(* IEC 61131-3 sources: volt/packages/volt-lsp-iec/test-corpus/bakon-nano/Device/Plc Logic/Application/Library Manager/(unresolved)/visu interfaces, 19 files *)

(* ---- RECIPE_FILEPARAMETERS.dut ---- *)
TYPE RECIPE_FILEPARAMETERS :
STRUCT
	PSTRECIPEDEFINITION : POINTER TO STRING;
	PSTRECIPE : POINTER TO STRING;
	PSTFILEPATH : POINTER TO STRING(512);
END_STRUCT
END_TYPE

(* ---- VISUSTRUCTCOLORSITF.dut ---- *)
TYPE VISUSTRUCTCOLORSITF :
STRUCT
	DWFRAMECOLOR : DWORD;
	DWFILLCOLOR : DWORD;
END_STRUCT
END_TYPE

(* ---- VISUSTRUCTELEMENTLOOKITF.dut ---- *)
TYPE VISUSTRUCTELEMENTLOOKITF :
STRUCT
	ILINEWIDTH : INT;
	DWFILLFLAGS : DWORD;
	DWFRAMEFLAGS : DWORD;
	WLINECAPFLAG : WORD;
	WLINEJOINFLAG : WORD;
	IMITERLIMIT : BYTE;
END_STRUCT
END_TYPE

(* ---- VISUSTRUCTPOINTITF.dut ---- *)
TYPE VISUSTRUCTPOINTITF :
STRUCT
	IX : INT;
	IY : INT;
END_STRUCT
END_TYPE

(* ---- VISUSTRUCTSIMPLERECTANGLEITF.dut ---- *)
TYPE VISUSTRUCTSIMPLERECTANGLEITF :
STRUCT
	PTTOPLEFT : VisuStructPointItf;
	PTBOTTOMRIGHT : VisuStructPointItf;
END_STRUCT
END_TYPE

(* ---- GVL.gvl ---- *)
VAR_GLOBAL
	G_VISUCOMMANDMANAGER : ICommandManager;
	G_VISUCOMMANDMANAGER2 : ICommandManager2;
	G_GLOBALCLIENTMANAGER : IVisuGlobalClientManager;
END_VAR

(* ---- GVL_CONSTANT.gvl ---- *)
VAR_GLOBAL
	VISU_INVALID_ID : INT := -1;
END_VAR

(* ---- IATTACHEDVISUALELEMENT.itf ---- *)
INTERFACE IATTACHEDVISUALELEMENT
END_INTERFACE

METHOD GETLOCATION : VisuStructSimpleRectangleItf
END_METHOD

(* ---- IBUTTONCLIENTSTATE.itf ---- *)
INTERFACE IBUTTONCLIENTSTATE
END_INTERFACE

METHOD ISPRESSED : BOOL
END_METHOD

METHOD SETPRESSED
VAR_INPUT
	BPRESSED : BOOL;
END_VAR
END_METHOD

(* ---- ICOMMANDMANAGER.itf ---- *)
INTERFACE ICOMMANDMANAGER
END_INTERFACE

METHOD GETCOMMAND : IGeneralCommand
VAR_INPUT
	IINDEX : INT;
END_VAR
END_METHOD

METHOD REGISTERCOMMAND : BOOL
VAR_INPUT
	CMD : IGeneralCommand;
END_VAR
END_METHOD

METHOD UNREGISTERCOMMAND : BOOL
VAR_INPUT
	CMD : IGeneralCommand;
END_VAR
END_METHOD

(* ---- ICOMMANDMANAGER2.itf ---- *)
INTERFACE ICOMMANDMANAGER2
END_INTERFACE

METHOD GETCOMMAND : IGeneralCommand2
VAR_INPUT
	IINDEX : INT;
END_VAR
END_METHOD

METHOD REGISTERCOMMAND : BOOL
VAR_INPUT
	CMD : IGeneralCommand2;
END_VAR
END_METHOD

METHOD UNREGISTERCOMMAND : BOOL
VAR_INPUT
	CMD : IGeneralCommand2;
END_VAR
END_METHOD

(* ---- IGENERALCOMMAND.itf ---- *)
INTERFACE IGENERALCOMMAND
END_INTERFACE

METHOD EXECUTE : DWORD
VAR_INPUT
	DWPARAM1 : DWORD;
	DWPARAM2 : DWORD;
END_VAR
END_METHOD

(* ---- IGENERALCOMMAND2.itf ---- *)
INTERFACE IGENERALCOMMAND2
END_INTERFACE

METHOD EXECUTE : __XWORD
VAR_INPUT
	DWPARAM1 : __XWORD;
	DWPARAM2 : __XWORD;
END_VAR
END_METHOD

(* ---- IGENERIC.itf ---- *)
INTERFACE IGENERIC
END_INTERFACE

METHOD GETINTERFACE : POINTER TO BYTE
VAR_INPUT
	DWITFID : DWORD;
END_VAR
END_METHOD

(* ---- IGLOBALCLIENTMANAGERLISTENER.itf ---- *)
INTERFACE IGLOBALCLIENTMANAGERLISTENER
END_INTERFACE

METHOD CLIENTCREATED
VAR_INPUT
	IGLOBALCLIENTID : INT;
	EVISUCLIENTTYPE : Visu_ClientTypeItf;
END_VAR
END_METHOD

METHOD CLIENTDESTROYED
VAR_INPUT
	IGLOBALCLIENTID : INT;
	EVISUCLIENTTYPE : Visu_ClientTypeItf;
END_VAR
END_METHOD

(* ---- IVISUGLOBALCLIENTMANAGER.itf ---- *)
INTERFACE IVISUGLOBALCLIENTMANAGER
END_INTERFACE

METHOD REGISTERORUPDATECLIENT : INT
VAR_INPUT
	IGLOBALCLIENTID : INT;
	EVISUCLIENTTYPE : Visu_ClientTypeItf;
END_VAR
END_METHOD

METHOD SETCURRENTCLIENTID : BOOL
VAR_INPUT
	IGLOBALCLIENTID : INT;
END_VAR
END_METHOD

(* ---- IVISUGLOBALCLIENTMANAGER2.itf ---- *)
INTERFACE IVISUGLOBALCLIENTMANAGER2
END_INTERFACE

METHOD ADDGLOBALCLIENTMANAGERLISTENER : BOOL
VAR_INPUT
	ITFGLOBALCLIENTMANAGERLISTENER : IGlobalClientManagerListener;
END_VAR
END_METHOD

(* ---- IVISUGLOBALCLIENTMANAGER3.itf ---- *)
INTERFACE IVISUGLOBALCLIENTMANAGER3
END_INTERFACE

METHOD UNREGISTERCLIENT : BOOL
VAR_INPUT
	IGLOBALCLIENTID : INT;
	EVISUCLIENTTYPE : Visu_ClientTypeItf;
END_VAR
END_METHOD

(* ---- VISU_CLIENTTYPEITF.dut ---- *)
TYPE VISU_CLIENTTYPEITF :
(
	UNKNOWN := 16#0,
	PROGRAMMINGSYSTEM := 16#1,
	STANDALONEVISUALIZATION := 16#2,
	TARGETVISUALIZATION := 16#4,
	WEBVISUALIZATION := 16#8,
	HMITARGETVISUALIZATION := 16#10,
	REMOTEVISUALIZATIONS := 16#1B,
	ALLVISUALIZATIONS := 16#1F
);
END_TYPE
